// TIA Portal V18 export
// export: Created 2026-06-13T06:09:35.6476296Z, ExportSetting WithDefaults, DisplayName Totally Integrated Automation Portal, DisplayVersion V18, DisplayName TIA Portal Openness, DisplayVersion V18, DisplayName TIA Portal Version Control Interface, DisplayVersion V18, DisplayName STEP 7 Professional, DisplayVersion V18, DisplayName STEP 7 Safety, DisplayVersion V18, DisplayName WinCC Professional, DisplayVersion V18
DATA_BLOCK "AI_Timers_PLC2"   // DB1
TITLE = AI_Timers_PLC2
{ S7_Optimized_Access := 'TRUE' }
VERSION : 0.1
// Global DB containing all timers and PID instances
// stored: AutoNumber true, DBAccessibleFromOPCUA true, IsOnlyStoredInLoadMemory false, IsRetainMemResEnabled false, IsWriteProtectedInAS false, MemoryReserve 100
   VAR
      AI_Timer_Dosing_Bon3 : IEC_TIMER;
      AI_Timer_Dosing_Bon4 : IEC_TIMER;
      AI_Timer_Khuay_Bon3 : IEC_TIMER;
      AI_Timer_Khuay_Thuan_Bon4 : IEC_TIMER;
      AI_Timer_Khuay_Nghich_Bon4 : IEC_TIMER;
      AI_Timer_Thanh_Trung_Bon4 : IEC_TIMER;
      AI_Timer_DryRun_Bon4 : IEC_TIMER;
      AI_Timer_Heartbeat_PLC2 : IEC_TIMER;
   END_VAR
BEGIN
END_DATA_BLOCK
